FUNCTION_BLOCK CarriageController
  (* Standard: 61499-2 *)
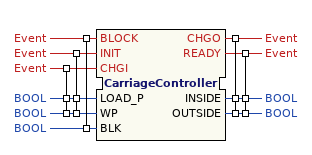
  EVENT_INPUT
    BLOCK WITH BLK;
    INIT WITH LOAD_P, WP;
    CHGI WITH LOAD_P, WP;
  END_EVENT
  EVENT_OUTPUT
    CHGO WITH INSIDE, OUTSIDE;
    READY WITH INSIDE, OUTSIDE;
  END_EVENT
  VAR_INPUT
    LOAD_P : BOOL;
    WP : BOOL;
    BLK : BOOL;
  END_VAR
  VAR_OUTPUT
    INSIDE : BOOL;
    OUTSIDE : BOOL;
  END_VAR
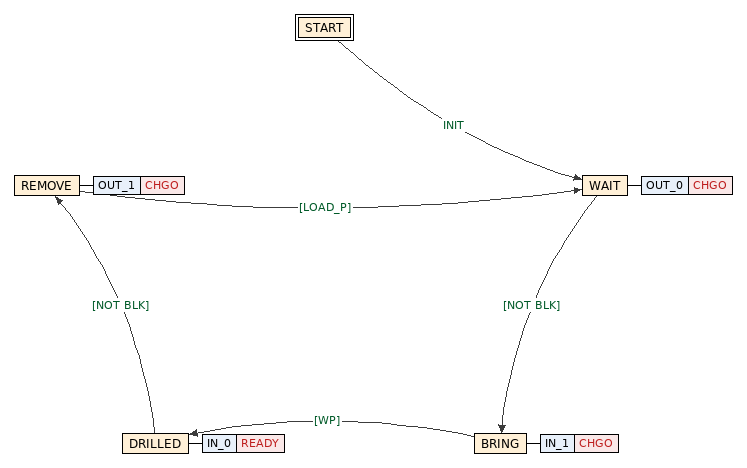
  EC_STATES
    START;
    WAIT : OUT_0 -> CHGO;
    BRING : IN_1 -> CHGO;
    DRILLED : IN_0 -> READY;
    REMOVE : OUT_1 -> CHGO;
  END_STATES
  EC_TRANSITIONS
    START TO WAIT := INIT;
    WAIT TO BRING := [NOT BLK];
    BRING TO DRILLED := [WP];
    DRILLED TO REMOVE := [NOT BLK];
    REMOVE TO WAIT := [LOAD_P];
  END_TRANSITIONS
  ALGORITHM IN_0 IN ST:
INSIDE := FALSE;&#10;
  END_ALGORITHM
  ALGORITHM IN_1 IN ST:
INSIDE := TRUE;&#10;
  END_ALGORITHM
  ALGORITHM OUT_0 IN ST:
OUTSIDE := FALSE;&#10;
  END_ALGORITHM
  ALGORITHM OUT_1 IN ST:
OUTSIDE := TRUE;&#10;
  END_ALGORITHM
END_FUNCTION_BLOCK
